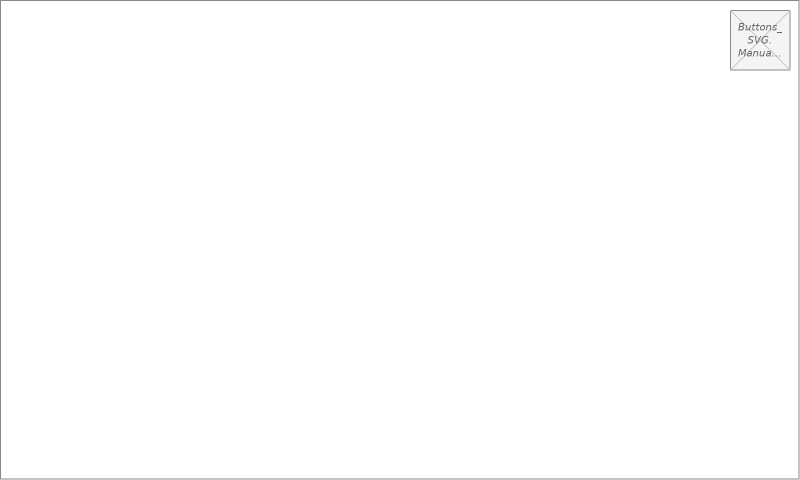
VISUALIZATION ManualButton_PNG  // 800x480
VAR_IN_OUT
	bCmdManual	: BOOL ; // switch to manual screen
END_VAR
    Image (730,10 60x60), image: Buttons_SVG.Manual mode Idle
        OnMouseClick: VisuUserMgmt Type=Login
        OnMouseClick: toggle bCmdManual
END_VISUALIZATION

(* stored: Version 1.1.0.1, ProductVersion 3.1.4024.5
   Visu ManualButton_PNG: Id {0d28c2e5-2aae-4d49-8380-e326fa839cb7} *)
